// SIMATIC S7-200 project (STEP 7-Micro/WIN), CPU 224 REL 02.01

ORGANIZATION_BLOCK MAIN:OB1
TITLE=PROGRAM COMMENTS
BEGIN
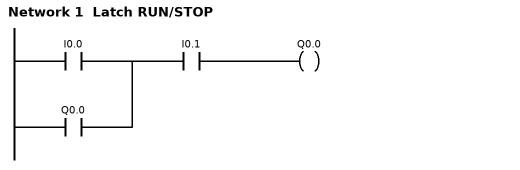
Network 1 // Latch RUN/STOP
LD     I0.0
O      Q0.0
A      I0.1
=      Q0.0
END_ORGANIZATION_BLOCK
